FUNCTION_BLOCK xswap_g
VAR_INPUT
    ix0: DINT;
    iy0: DINT;
END_VAR
VAR_IN_OUT
    x: ARRAY [0..29] OF LREAL;
END_VAR
VAR_TEMP
    temp: LREAL;
    k: DINT;
    temp_tmp: DINT;
    tmp: DINT;
END_VAR

FOR k := 0 TO 5 DO 
    temp_tmp := (ix0 + k) - 1;
    temp := x[temp_tmp];
    tmp := (iy0 + k) - 1;
    x[temp_tmp] := x[tmp];
    x[tmp] := temp;
END_FOR;

END_FUNCTION_BLOCK

(* stored: Version 1.1.0.1, ProductVersion 3.1.4024.12
   POU xswap_g: Id {be824ae0-713f-43c1-97b2-6baa4d940f16}, SpecialFunc None *)
